FUNCTION_BLOCK LinearClearLinkMC EXTENDS FBA_LinearTrifecta IMPLEMENTS I_EncodedDrive
VAR_OUTPUT
	pulse AT %Q* : INT;
	brakeRelease AT %Q* : BOOL := TRUE;
	enable : BOOL;
	A : BOOL;
	B : BOOL;
	clear : BOOL;
END_VAR
VAR	
	hlfb AT %I* : REAL := -9999; //high level feedback, if -9999 then servo is idle
	
	outputRegister AT %Q* : INT;
	pulseRequest : INT;
	
	homingDelay : TON;
	resetPulse : TP;
	
	mode : (HOLD, TARGET, CONTINUOUS, RESET_ERR);
	calculation : (IDLE, DOWN, UP, CALCULATE, DONE);
	maxPosition : LREAL;
	
	position, targetPos : LREAL;
	
	pulsePosition : INT;
	pulseCounter : INT;
	rotationsPerPulse : INT; //revolutions per pulse
	displacementPerPulse : LREAL; //displacement per pulse
END_VAR
VAR_STAT CONSTANT
	resetWidth : TIME := T#500MS;
	delayWidth : TIME := T#500MS;
END_VAR
VAR //constructor
	homingDirectionOut : BOOL; 			//homing direction - see <A>
	minPosition : LREAL;
	displacementPerRotation : LREAL; 	//displacement per revolution	
	unitsPerPulse : INT := 800; 		//800 Teknic units per rotation - default setting is 800 units (1 rotation) per pulse
END_VAR

//M-connector output register
outputRegister.0 := enable AND bEnable; 	//enable
outputRegister.1 := A; 						//direction bit - T = outwards, F = inwards
outputRegister.2 := B; 						//homing bit - after startup, set to TRUE to begin homing, then set to FALSE to finish homing
outputRegister.3 := clear; 					//reset bit

rotationsPerPulse := unitsPerPulse/800; //Teknic constant - 800 units per rotation
displacementPerPulse := displacementPerRotation * rotationsPerPulse;

resetPulse(IN:= , PT:= resetWidth, Q=> clear, ET=> ); //reset pulse

IF NOT enable AND NOT AtInnerLimit THEN
	homingComplete := FALSE;
	step := Homing.IDLE;
	mode := HOLD;
END_IF

override();

CASE mode OF		
	HOLD: //hold current position, no motion
		pulse := 0;
		pulseRequest := 0;
	
	TARGET:	//target a given position
		
		IF WithinTolerance(position, targetPos, displacementPerPulse) THEN
			pulseRequest := 0;
			pulse := 0;
			mode := HOLD;
			
		ELSIF NOT Active THEN
			A :=  position < targetPos;
			(*
			2 options to traverse to a target position:
				a)  send all pulses at once - continuous motion but may exceed limits, check for bounds before setting
				b)  1 pulse at a time - choppy but safer
			*)
			targetPos := MAX(targetPos, minPosition); //if below minPosition, set to minPosition
			targetPos := MIN(targetPos, maxPosition); //if above maxPosition, set to maxPosition
			
			pulseRequest := TO_INT(ABS(position - targetPos)/displacementPerPulse);
			//pulseRequest := 1;
		END_IF
		
	CONTINUOUS: //single pulses in the direction specified by moveContinuous()
		pulseRequest := 1;
		
	RESET_ERR: //reset pulse, servo may need to be rehomed aftewards
		pulse := 0;
		pulseRequest := 0;
		resetPulse.IN := TRUE;
		
		IF resetPulse.Q THEN
			resetPulse.IN := FALSE;
			mode := HOLD;
		END_IF
		
END_CASE

sequence();

PROPERTY Active : BOOL
GET
Active := hlfb <> -9999;
END_GET
END_PROPERTY

{attribute 'monitoring':='call'}
PROPERTY AtOuterLimit : BOOL
GET
AtOuterLimit := outerLimit <> limitSensorDefaultState;
END_GET
END_PROPERTY

METHOD PRIVATE calculatePositions : BOOL
(*
the purpose of this method is calculate the position at the outer limit

complete a full range traverse while counting the pulses, then multiply
	displacement per rotation
	rotations per pulse
	number of pulses for the traversal
and add to position at inner limit to get position at outer limit
*)
CASE calculation OF
	IDLE:
		calculation := DOWN;
		
	DOWN:
		moveContinuous(direction := MC_Negative_Direction);
		IF AtInnerLimit THEN
			calculation := UP;
			pulseCounter := 0;
		END_IF
		
	UP:
		moveContinuous(direction := MC_Positive_Direction);
		IF AtHome THEN
			maxPosition := minPosition + (displacementPerRotation * rotationsPerPulse * pulseCounter);
			calculation := DONE;
		END_IF
		
	DONE:
		calculation := 0;
		calculatePositions := TRUE;
		
END_CASE
END_METHOD

PROPERTY CurrentPosition : LREAL
GET
CurrentPosition := position;

//CurrentPosition := pulsePosition * displacementPerPulse;
END_GET
SET
position := CurrentPosition;
END_SET
END_PROPERTY

PROPERTY Error : BOOL
GET
END_GET
END_PROPERTY

METHOD homingSequence : BOOL
homingDelay(IN:= , PT:= delayWidth, Q=> , ET=> );

CASE step OF
	Homing.IDLE:
		enable := TRUE;
		A := FALSE;
		B := TRUE;
		brakeRelease := TRUE;
		
		homingComplete := FALSE;
		
		homingDelay.IN := TRUE;
		IF homingDelay.Q THEN
			homingDelay.IN := FALSE;
			//step := Homing.START;
			step := Homing.RETRY;
		END_IF
		
	Homing.START:
		IF homingDelay.Q THEN
			homingDelay.IN := FALSE;
			step := Homing.SET;
			
		ELSIF AtHome THEN
			homingDelay.IN := TRUE;
			
		ELSIF AtOuterLimit THEN
			step := Homing.RETRY;
		
		ELSE
			enable := TRUE;
			A := FALSE;
			B := TRUE;
			brakeRelease := TRUE;
		
		END_IF
	
	Homing.RETRY:
		IF AtInnerLimit THEN
			homingDelay.IN := TRUE;
			enable := FALSE;
			
			IF homingDelay.Q THEN
				homingDelay.IN := FALSE;
				step := Homing.START;
			END_IF
			
		ELSE
			enable := TRUE;
			A := FALSE;
			B := FALSE;
			brakeRelease := TRUE;
			
			mode := CONTINUOUS;
		END_IF

	Homing.SET:
		enable := TRUE;
		A := FALSE;
		B := FALSE;
		brakeRelease := TRUE;
		
		IF calculatePositions() THEN
			step := Homing.DONE;
		END_IF
		
	Homing.DONE:
		homingSequence := homingComplete := TRUE;
		
		pulsePosition := 0;
		
		mode := HOLD;
		step := Homing.IDLE;
	
END_CASE
END_METHOD

{attribute 'TcRpcEnable'}
METHOD moveAbsolute : BOOL
VAR_INPUT
	newTarget : LREAL;
END_VAR
IF target >= maxPosition AND target <= minPosition THEN
	A :=  position < targetPos;
	targetPos := newTarget;
	mode := TARGET;
	
	moveAbsolute := TRUE;
END_IF
END_METHOD

{attribute 'TcRpcEnable'}
METHOD moveContinuous : BOOL
VAR_INPUT
	direction : MC_Direction;
END_VAR
IF direction = MC_Negative_Direction THEN
	A := FALSE;
ELSIF direction = MC_Positive_Direction THEN
	A := TRUE;
END_IF

mode := CONTINUOUS;
END_METHOD

{attribute 'TcRpcEnable'}
METHOD moveRelative : BOOL
VAR_INPUT
	distance : LREAL;
END_VAR
targetPos := targetPos + distance;

mode := TARGET;
END_METHOD

METHOD PRIVATE override : BOOL
VAR_INPUT
END_VAR
(*
allowable motion is between AtHome and AtInnerLimit
*)
IF AtHome AND NOT Active THEN
	IF homingDirectionOut THEN //homing is outwards
		position := maxPosition;
		pulsePosition := pulseCounter;
	ELSE
		position := minPosition;
		pulsePosition := 0;
	END_IF
	

ELSIF AtInnerLimit AND NOT Active THEN
	IF homingDirectionOut THEN //homing is outwards
		position := minPosition;
		pulsePosition := 0;
	ELSE
		position := maxPosition;
		pulsePosition := pulseCounter;
	END_IF
END_IF

CASE mode OF		
	HOLD:
		//
	
	TARGET:
		IF
			(AtHome AND TargetPosition > CurrentPosition) OR
			(AtInnerLimit AND TargetPosition > CurrentPosition) OR
			(AtOuterLimit AND TargetPosition < CurrentPosition)
		THEN
			mode := HOLD;
		END_IF
		
	CONTINUOUS:
		IF
			(AtHome AND A) OR
			(AtInnerLimit AND A) OR
			(AtOuterLimit AND NOT A)
		THEN
			mode := HOLD;
		END_IF
		
	RESET_ERR:
		//
		
END_CASE
END_METHOD

METHOD reset : BOOL
VAR_INPUT
END_VAR
mode := RESET_ERR;
END_METHOD

METHOD PRIVATE sequence : BOOL
VAR_INPUT
END_VAR
IF Active THEN //servo is active
	IF A THEN //positive direction
		position := position + (displacementPerPulse * pulse);
		pulsePosition := pulsePosition + pulse;
		
		pulseCounter := pulseCounter + pulse;
	ELSE //negative direction
		position := position - (displacementPerPulse * pulse);
		pulsePosition := pulsePosition - pulse;
		
		pulseCounter := pulseCounter - pulse;
	END_IF
	pulse := 0; //pulses already received, can be set to 0 so position change is not compounded

ELSIF pulse = 0 THEN //servo is not active
	pulse := pulseRequest;
END_IF

pulseRequest := 0; //remove this if not working as intended
END_METHOD

METHOD stop : BOOL
VAR_INPUT
END_VAR
mode := HOLD;
END_METHOD

PROPERTY TargetPosition : LREAL
GET
END_GET
SET
targetPos := TargetPosition;
END_SET
END_PROPERTY

METHOD toHome : BOOL
VAR_INPUT
END_VAR
IF homingDirectionOut THEN
	moveAbsolute(newTarget := maxPosition);
ELSE
	moveAbsolute(newTarget := minPosition);
END_IF
END_METHOD

END_FUNCTION_BLOCK

(* stored: Version 1.1.0.1, ProductVersion 3.1.4024.11
   POU LinearClearLinkMC: Id {525d7a58-b099-4630-95c5-878d2c9eeac9}, SpecialFunc None
   Folder Private: Id {28dbda7f-e8e4-4cd0-ad26-239756599ef1}
   Folder Properties: Id {53fb867d-2749-435b-87c7-45fe10aac940}
   Property Active: Id {f96e1f9d-9991-4651-a575-cb341e2d8ea3}
   Get Get: Id {bc44c60a-a027-4357-b941-a5a35bd2ac9b}
   Property AtOuterLimit: Id {79da769f-f6e6-4af2-b32c-ad787d5b12d0}
   Get Get: Id {606d01cc-509e-409e-bb50-85d8fd1f1f02}
   Method calculatePositions: Id {a02964bb-645c-4e49-9dbf-5290a643a91f}
   Property CurrentPosition: Id {6986f970-ba1e-4d4d-b9d3-12404339f870}
   Get Get: Id {8d42d596-9590-4b6a-be1f-b4eae8cfe681}
   Set Set: Id {f741cae1-d13a-48ba-b5ca-ce8ace500b9e}
   Property Error: Id {09047c6a-d518-4f8a-bc5c-aa7de353f004}
   Get Get: Id {2b5d5f4b-ee4b-4695-aad2-0b5305ee2133}
   Method homingSequence: Id {2eaeec5a-2ba5-4b28-b338-e8a91d3c1693}
   Method moveAbsolute: Id {007bb13e-56f5-474c-9b07-aaeaaccc18d8}
   Method moveContinuous: Id {0763384e-b190-47a7-823a-1e8114cb94f4}
   Method moveRelative: Id {109d4c5d-cb0f-4f62-b291-68b4c84415db}
   Method override: Id {4fd8c0d6-b728-4f86-9142-ee32bcc08d3e}
   Method reset: Id {d73d50c4-6d4e-4efe-99ae-f87e9c32e3a0}
   Method sequence: Id {fabcde92-2d7e-47e1-82f8-d0cfcb9e9f9a}
   Method stop: Id {5d2f6a07-7ceb-4538-b22e-bf46aa71ac3a}
   Property TargetPosition: Id {d105dc41-bb9b-42a5-b821-71a06002d4c7}
   Get Get: Id {5158b650-db12-4232-a887-111b26684f14}
   Set Set: Id {8b3607e5-acdb-4414-aec8-5e953cf74ea6}
   Method toHome: Id {aa05bb74-3208-4665-940d-96e24df22079} *)
